// TIA Portal V17 export
// export: Created 2024-09-03T21:55:03.1361635Z, ExportSetting WithDefaults, DisplayName Totally Integrated Automation Portal, DisplayVersion V17 Update 7, DisplayName TIA Portal Openness, DisplayVersion V17 Update 7, DisplayName TIA Portal Version Control Interface, DisplayVersion V17, DisplayName SINAMICS Startdrive Advanced, DisplayVersion V17 SP2, DisplayName SINAMICS Startdrive G110M, G120, G120C, G120D, G120P, G115D, DisplayVersion V17 SP2, DisplayName SINAMICS Startdrive G130, G150, S120, S150, SINAMICS MV, S210, DisplayVersion V17 SP2, DisplayName STEP 7 Professional, DisplayVersion V17 Update 7, DisplayName STEP 7 Safety, DisplayVersion V17 Update 6, DisplayName WinCC Advanced / Unified PC, DisplayVersion V17 Update 7
VAR_GLOBAL   // PLC tag table "Turn table"
   iTurnTableInputs AT %IW300 : Word;
   qTurnTableOutputs AT %QW300 : Word;
   iTurnTableOperating AT %I300.4 : Bool;
   iTurnTableIndexerInPosition AT %I300.5 : Bool;
   qTurnTableStop AT %Q300.1 : Bool;
   qTurnTableCycleCW AT %Q300.2 : Bool;
   qTurnTableCycleCCW AT %Q300.3 : Bool;
   qTurnTableCycleJogCW AT %Q300.4 : Bool;
   qTurnTableCycleJogCCW AT %Q300.5 : Bool;
END_VAR
